// TIA Portal project "Comparadores" (V16)

(* hardware
DEVICE "S7-1200 station_1"  S7-1200 Station
   slot 0: "Rack_0"  S7-1200 Rack  Rack  V1.0
   slot 1: "PLC_1"  CPU 1214C AC/DC/Rly  6ES7 214-1BG40-0XB0  V4.4
*)

// ===== PLC "PLC_1"  CPU 1214C AC/DC/Rly =====

VAR_GLOBAL   // PLC tag table "Tabla de variables estándar"
   ""INT TMP"" AT %I0.0 : Bool;
   ""INT CU"" AT %I0.1 : Bool;
   ""INT CD"" AT %I0.2 : Bool;
   ""INT RESET UP"" AT %I0.3 : Bool;
   ""INT RESET DOWN"" AT %I0.4 : Bool;
   ""CONTACTO NC"" AT %I0.5 : Bool;
   ""Tag_2"" AT %Q0.0 : Bool;
   ""Tag_3"" AT %Q0.1 : Bool;
   ""Tag_1"" AT %Q0.2 : Bool;
   ""Tag_4"" AT %Q0.3 : Bool;
   ""Tag_5"" AT %Q0.4 : Bool;
   ""Tag_6"" AT %Q0.5 : Bool;
   ""Tag_7"" AT %Q0.6 : Bool;
   ""Tag_10"" AT %Q0.7 : Bool;
   ""Tag_11"" AT %Q1.0 : Bool;
END_VAR